TYPE E_MoMaStates :
(
	Init,
	Prepare,
	Moving_TM,
	Moving_LD,
	Succeeded, 
	Failed,
	ServiceNeeded
)UDINT;
END_TYPE

(* stored: Version 1.1.0.1, ProductVersion 3.1.4024.11
   DUT E_MoMaStates: Id {10ce00cc-d7fa-4567-a974-ec2e7a693170} *)
